(* IEC 61131-3 sources: Antarbhukti-LLM/DatasetCreation/UpgradesGeneration/test_batch, 10 files *)

(* ---- ACTUATOR_2P_sfc_iter_01_L2_iter_01_upgraded.st ---- *)
PROGRAM SFC_Program
(* Auto-generated by SFCJSONConverter *)

VAR
  InitCycle_active : BOOL := FALSE;
  SafetyCheckInput_active : BOOL := FALSE;
  SafetyError_active : BOOL := FALSE;
  Branch_0_active : BOOL := FALSE;
  Branch_1_active : BOOL := FALSE;
  Branch_2_active : BOOL := FALSE;
  Step_255_active : BOOL := FALSE;
  ApplyOutput_active : BOOL := FALSE;
  TimeoutSafeStop_active : BOOL := FALSE;
  SafetyLog_active : BOOL := FALSE;
  IN : INT := 0;
  TEST : INT := 0;
  ARE : INT := 0;
  CYCLE_TIME : TIME := T#0s;
  SENS : INT := 0;
  SELF_ACT_TIME : TIME := T#0s;
  SELF_ACT_PULSE : TIME := T#0s;
  SELF_ACT_CYCLES : INT := 0;
  OUT : BOOL := FALSE;
  ARO : BOOL := FALSE;
  ARX : INT := 0;
  timer : TIMER;
  pwgen : PWGEN;
  INPUT_VALID : BOOL := FALSE;
  SAFETY_ERROR_FLAG : BOOL := FALSE;
  SAFETY_ERROR_CODE : UINT := 0;
  CUMULATIVE_CYCLE_TIME : TIME := T#0s;
  MAX_SAFE_CYCLE_TIME : TIME := T#0s;
  TIMEOUT_EXCEEDED : BOOL := FALSE;
  TIMEOUT_ERROR_FLAG : BOOL := FALSE;
  TIMEOUT_LOG_TIME : TIME := T#0s;
  SAFETY_LOG_CODE : UINT := 0;
  TIMEOUT_LOG_CODE : UINT := 0;
  LOGGED_CYCLE_TIME : TIME := T#0s;
END_VAR

(* --- Initialize initial step --- *)
IF NOT InitCycle_active THEN
  InitCycle_active := TRUE;
END_IF;

(* --- Step actions --- *)
IF InitCycle_active THEN
  timer(trun := MUL_T_AI(SELF_ACT_PULSE,2 * SELF_ACT_CYCLES), toff := SELF_ACT_TIME, Test := TEST, ARE := ARE, arx := ARX); ARX := timer.ARX; ARO := timer.ARO;
END_IF;
IF SafetyCheckInput_active THEN
  INPUT_VALID := (IN >= BYTE#0) AND (IN <= BYTE#255) AND (SENS > BYTE#0) AND (SENS <= BYTE#255); CUMULATIVE_CYCLE_TIME := CUMULATIVE_CYCLE_TIME + CYCLE_TIME;
END_IF;
IF SafetyError_active THEN
  out := FALSE; SAFETY_ERROR_FLAG := TRUE; SAFETY_ERROR_CODE := UINT#1001;
END_IF;
IF Branch_0_active THEN
  pwgen(PTL := SELF_ACT_PULSE, PTH := SELF_ACT_PULSE); out := pwgen.Q;
END_IF;
IF Branch_1_active THEN
  out := FALSE;
END_IF;
IF Branch_2_active THEN
  out := TRUE;
END_IF;
IF Step_255_active THEN
  pwgen.PTH := (CYCLE_TIME * BYTE_TO_TIME(BAND_B(IN,SENS)) ) / BYTE_TO_TIME(BYTE#255); pwgen.PTL := CYCLE_TIME - pwgen.PTH; pwgen(); out := pwgen.Q;
END_IF;
IF ApplyOutput_active THEN
  TIMEOUT_EXCEEDED := CUMULATIVE_CYCLE_TIME > MAX_SAFE_CYCLE_TIME;
END_IF;
IF TimeoutSafeStop_active THEN
  out := FALSE; TIMEOUT_ERROR_FLAG := TRUE; TIMEOUT_LOG_TIME := CUMULATIVE_CYCLE_TIME; CUMULATIVE_CYCLE_TIME := T#0s;
END_IF;
IF SafetyLog_active THEN
  SAFETY_LOG_CODE := SAFETY_ERROR_CODE; TIMEOUT_LOG_CODE := TIMEOUT_ERROR_FLAG; LOGGED_CYCLE_TIME := CUMULATIVE_CYCLE_TIME;
END_IF;

(* --- Transitions --- *)
IF InitCycle_active AND (TRUE) THEN
  InitCycle_active := FALSE;
  SafetyCheckInput_active := TRUE;
END_IF;
IF SafetyCheckInput_active AND (INPUT_VALID = FALSE) THEN
  SafetyCheckInput_active := FALSE;
  SafetyError_active := TRUE;
END_IF;
IF SafetyCheckInput_active AND (INPUT_VALID = TRUE AND aro = TRUE) THEN
  SafetyCheckInput_active := FALSE;
  Branch_0_active := TRUE;
END_IF;
IF SafetyCheckInput_active AND (INPUT_VALID = TRUE AND aro = FALSE AND in<sens) THEN
  SafetyCheckInput_active := FALSE;
  Branch_1_active := TRUE;
END_IF;
IF SafetyCheckInput_active AND (INPUT_VALID = TRUE AND aro = FALSE AND NOT (in<sens) AND BYTE_TO_USINT(in)>USINT#255-BYTE_TO_USINT(sens)) THEN
  SafetyCheckInput_active := FALSE;
  Branch_2_active := TRUE;
END_IF;
IF SafetyCheckInput_active AND (INPUT_VALID = TRUE AND aro = FALSE AND NOT (in<sens) AND NOT (BYTE_TO_USINT(in)>USINT#255-BYTE_TO_USINT(sens))) THEN
  SafetyCheckInput_active := FALSE;
  Step_255_active := TRUE;
END_IF;
IF Branch_0_active AND (TRUE) THEN
  Branch_0_active := FALSE;
  ApplyOutput_active := TRUE;
END_IF;
IF Branch_1_active AND (TRUE) THEN
  Branch_1_active := FALSE;
  ApplyOutput_active := TRUE;
END_IF;
IF Branch_2_active AND (TRUE) THEN
  Branch_2_active := FALSE;
  ApplyOutput_active := TRUE;
END_IF;
IF Step_255_active AND (TRUE) THEN
  Step_255_active := FALSE;
  ApplyOutput_active := TRUE;
END_IF;
IF ApplyOutput_active AND (TIMEOUT_EXCEEDED = TRUE) THEN
  ApplyOutput_active := FALSE;
  TimeoutSafeStop_active := TRUE;
END_IF;
IF ApplyOutput_active AND (TIMEOUT_EXCEEDED = FALSE) THEN
  ApplyOutput_active := FALSE;
  InitCycle_active := TRUE;
END_IF;
IF TimeoutSafeStop_active AND (TRUE) THEN
  TimeoutSafeStop_active := FALSE;
  SafetyLog_active := TRUE;
END_IF;
IF SafetyError_active AND (TRUE) THEN
  SafetyError_active := FALSE;
  SafetyLog_active := TRUE;
END_IF;
IF SafetyLog_active AND (TRUE) THEN
  SafetyLog_active := FALSE;
  InitCycle_active := TRUE;
END_IF;

END_PROGRAM

(* ---- ACTUATOR_2P_sfc_iter_01_L2_iter_02_upgraded.st ---- *)
PROGRAM SFC_Program
(* Auto-generated by SFCJSONConverter *)

VAR
  InitCycle_active : BOOL := FALSE;
  SafetyCheckInput_active : BOOL := FALSE;
  SafetyError_active : BOOL := FALSE;
  SafetyLog_Error_active : BOOL := FALSE;
  Branch_0_active : BOOL := FALSE;
  Branch_1_active : BOOL := FALSE;
  Branch_2_active : BOOL := FALSE;
  Step_255_active : BOOL := FALSE;
  ApplyOutput_active : BOOL := FALSE;
  TimeoutSafeStop_active : BOOL := FALSE;
  SafetyLog_Timeout_active : BOOL := FALSE;
  IN : INT := 0;
  TEST : INT := 0;
  ARE : INT := 0;
  CYCLE_TIME : TIME := T#0s;
  SENS : INT := 0;
  SELF_ACT_TIME : TIME := T#0s;
  SELF_ACT_PULSE : TIME := T#0s;
  SELF_ACT_CYCLES : INT := 0;
  OUT : BOOL := FALSE;
  ARO : BOOL := FALSE;
  ARX : INT := 0;
  timer : TIMER;
  pwgen : PWGEN;
  INPUT_VALID : BOOL := FALSE;
  SAFETY_ERROR_FLAG : BOOL := FALSE;
  SAFETY_ERROR_CODE : UINT := 0;
  CUMULATIVE_CYCLE_TIME : TIME := T#0s;
  MAX_SAFE_CYCLE_TIME : TIME := T#0s;
  TIMEOUT_EXCEEDED : BOOL := FALSE;
  TIMEOUT_ERROR_FLAG : BOOL := FALSE;
  TIMEOUT_LOG_TIME : TIME := T#0s;
  SAFETY_LOG_CODE : UINT := 0;
  SAFETY_LOG_TIME : TIME := T#0s;
  SAFETY_LOG_IN : INT := 0;
  SAFETY_LOG_SENS : INT := 0;
END_VAR

(* --- Initialize initial step --- *)
IF NOT InitCycle_active THEN
  InitCycle_active := TRUE;
END_IF;

(* --- Step actions --- *)
IF InitCycle_active THEN
  timer(trun := MUL_T_AI(SELF_ACT_PULSE,2 * SELF_ACT_CYCLES), toff := SELF_ACT_TIME, Test := TEST, ARE := ARE, arx := ARX); ARX := timer.ARX; ARO := timer.ARO;
END_IF;
IF SafetyCheckInput_active THEN
  INPUT_VALID := (IN >= BYTE#0) AND (IN <= BYTE#255) AND (SENS > BYTE#0) AND (SENS <= BYTE#255); CUMULATIVE_CYCLE_TIME := CUMULATIVE_CYCLE_TIME + CYCLE_TIME;
END_IF;
IF SafetyError_active THEN
  out := FALSE; SAFETY_ERROR_FLAG := TRUE; SAFETY_ERROR_CODE := UINT#1001;
END_IF;
IF SafetyLog_Error_active THEN
  SAFETY_LOG_CODE := SAFETY_ERROR_CODE; SAFETY_LOG_TIME := CUMULATIVE_CYCLE_TIME; SAFETY_LOG_IN := IN; SAFETY_LOG_SENS := SENS;
END_IF;
IF Branch_0_active THEN
  pwgen(PTL := SELF_ACT_PULSE, PTH := SELF_ACT_PULSE); out := pwgen.Q;
END_IF;
IF Branch_1_active THEN
  out := FALSE;
END_IF;
IF Branch_2_active THEN
  out := TRUE;
END_IF;
IF Step_255_active THEN
  pwgen.PTH := (CYCLE_TIME * BYTE_TO_TIME(BAND_B(IN,SENS)) ) / BYTE_TO_TIME(BYTE#255); pwgen.PTL := CYCLE_TIME - pwgen.PTH; pwgen(); out := pwgen.Q;
END_IF;
IF ApplyOutput_active THEN
  TIMEOUT_EXCEEDED := CUMULATIVE_CYCLE_TIME > MAX_SAFE_CYCLE_TIME;
END_IF;
IF TimeoutSafeStop_active THEN
  out := FALSE; TIMEOUT_ERROR_FLAG := TRUE; TIMEOUT_LOG_TIME := CUMULATIVE_CYCLE_TIME; CUMULATIVE_CYCLE_TIME := T#0s;
END_IF;
IF SafetyLog_Timeout_active THEN
  SAFETY_LOG_CODE := UINT#2001; SAFETY_LOG_TIME := TIMEOUT_LOG_TIME;
END_IF;

(* --- Transitions --- *)
IF InitCycle_active AND (TRUE) THEN
  InitCycle_active := FALSE;
  SafetyCheckInput_active := TRUE;
END_IF;
IF SafetyCheckInput_active AND (INPUT_VALID = FALSE) THEN
  SafetyCheckInput_active := FALSE;
  SafetyError_active := TRUE;
END_IF;
IF SafetyCheckInput_active AND (INPUT_VALID = TRUE AND aro = TRUE) THEN
  SafetyCheckInput_active := FALSE;
  Branch_0_active := TRUE;
END_IF;
IF SafetyCheckInput_active AND (INPUT_VALID = TRUE AND aro = FALSE AND in<sens) THEN
  SafetyCheckInput_active := FALSE;
  Branch_1_active := TRUE;
END_IF;
IF SafetyCheckInput_active AND (INPUT_VALID = TRUE AND aro = FALSE AND NOT (in<sens) AND BYTE_TO_USINT(in)>USINT#255-BYTE_TO_USINT(sens)) THEN
  SafetyCheckInput_active := FALSE;
  Branch_2_active := TRUE;
END_IF;
IF SafetyCheckInput_active AND (INPUT_VALID = TRUE AND aro = FALSE AND NOT (in<sens) AND NOT (BYTE_TO_USINT(in)>USINT#255-BYTE_TO_USINT(sens))) THEN
  SafetyCheckInput_active := FALSE;
  Step_255_active := TRUE;
END_IF;
IF Branch_0_active AND (TRUE) THEN
  Branch_0_active := FALSE;
  ApplyOutput_active := TRUE;
END_IF;
IF Branch_1_active AND (TRUE) THEN
  Branch_1_active := FALSE;
  ApplyOutput_active := TRUE;
END_IF;
IF Branch_2_active AND (TRUE) THEN
  Branch_2_active := FALSE;
  ApplyOutput_active := TRUE;
END_IF;
IF Step_255_active AND (TRUE) THEN
  Step_255_active := FALSE;
  ApplyOutput_active := TRUE;
END_IF;
IF ApplyOutput_active AND (TIMEOUT_EXCEEDED = TRUE) THEN
  ApplyOutput_active := FALSE;
  TimeoutSafeStop_active := TRUE;
END_IF;
IF ApplyOutput_active AND (TIMEOUT_EXCEEDED = FALSE) THEN
  ApplyOutput_active := FALSE;
  InitCycle_active := TRUE;
END_IF;
IF TimeoutSafeStop_active AND (TRUE) THEN
  TimeoutSafeStop_active := FALSE;
  SafetyLog_Timeout_active := TRUE;
END_IF;
IF SafetyLog_Timeout_active AND (TRUE) THEN
  SafetyLog_Timeout_active := FALSE;
  InitCycle_active := TRUE;
END_IF;
IF SafetyError_active AND (TRUE) THEN
  SafetyError_active := FALSE;
  SafetyLog_Error_active := TRUE;
END_IF;
IF SafetyLog_Error_active AND (TRUE) THEN
  SafetyLog_Error_active := FALSE;
  SafetyLog_Error_active := TRUE;
END_IF;

END_PROGRAM

(* ---- ACTUATOR_2P_sfc_iter_01_L2_iter_03_upgraded.st ---- *)
PROGRAM SFC_Program
(* Auto-generated by SFCJSONConverter *)

VAR
  InitCycle_active : BOOL := FALSE;
  SafetyCheckInput_active : BOOL := FALSE;
  SafetyLog_active : BOOL := FALSE;
  SafetyError_active : BOOL := FALSE;
  SafetyErrorLog_active : BOOL := FALSE;
  Branch_0_active : BOOL := FALSE;
  Branch_1_active : BOOL := FALSE;
  Branch_2_active : BOOL := FALSE;
  Step_255_active : BOOL := FALSE;
  ApplyOutput_active : BOOL := FALSE;
  TimeoutSafeStop_active : BOOL := FALSE;
  IN : INT := 0;
  TEST : INT := 0;
  ARE : INT := 0;
  CYCLE_TIME : TIME := T#0s;
  SENS : INT := 0;
  SELF_ACT_TIME : TIME := T#0s;
  SELF_ACT_PULSE : TIME := T#0s;
  SELF_ACT_CYCLES : INT := 0;
  OUT : BOOL := FALSE;
  ARO : BOOL := FALSE;
  ARX : INT := 0;
  timer : TIMER;
  pwgen : PWGEN;
  INPUT_VALID : BOOL := FALSE;
  SAFETY_ERROR_FLAG : BOOL := FALSE;
  SAFETY_ERROR_CODE : UINT := 0;
  CUMULATIVE_CYCLE_TIME : TIME := T#0s;
  MAX_SAFE_CYCLE_TIME : TIME := T#0s;
  TIMEOUT_EXCEEDED : BOOL := FALSE;
  TIMEOUT_ERROR_FLAG : BOOL := FALSE;
  TIMEOUT_LOG_TIME : TIME := T#0s;
  SAFETY_LOG_IN : INT := 0;
  SAFETY_LOG_SENS : INT := 0;
  SAFETY_LOG_CUMULATIVE_TIME : TIME := T#0s;
  SAFETY_ERROR_LOG_CODE : UINT := 0;
  SAFETY_ERROR_LOG_TIME : TIME := T#0s;
END_VAR

(* --- Initialize initial step --- *)
IF NOT InitCycle_active THEN
  InitCycle_active := TRUE;
END_IF;

(* --- Step actions --- *)
IF InitCycle_active THEN
  timer(trun := MUL_T_AI(SELF_ACT_PULSE,2 * SELF_ACT_CYCLES), toff := SELF_ACT_TIME, Test := TEST, ARE := ARE, arx := ARX); ARX := timer.ARX; ARO := timer.ARO;
END_IF;
IF SafetyCheckInput_active THEN
  INPUT_VALID := (IN >= BYTE#0) AND (IN <= BYTE#255) AND (SENS > BYTE#0) AND (SENS <= BYTE#255); CUMULATIVE_CYCLE_TIME := CUMULATIVE_CYCLE_TIME + CYCLE_TIME;
END_IF;
IF SafetyLog_active THEN
  SAFETY_LOG_IN := IN; SAFETY_LOG_SENS := SENS; SAFETY_LOG_CUMULATIVE_TIME := CUMULATIVE_CYCLE_TIME;
END_IF;
IF SafetyError_active THEN
  out := FALSE; SAFETY_ERROR_FLAG := TRUE; SAFETY_ERROR_CODE := UINT#1001;
END_IF;
IF SafetyErrorLog_active THEN
  SAFETY_ERROR_LOG_CODE := SAFETY_ERROR_CODE; SAFETY_ERROR_LOG_TIME := CUMULATIVE_CYCLE_TIME;
END_IF;
IF Branch_0_active THEN
  pwgen(PTL := SELF_ACT_PULSE, PTH := SELF_ACT_PULSE); out := pwgen.Q;
END_IF;
IF Branch_1_active THEN
  out := FALSE;
END_IF;
IF Branch_2_active THEN
  out := TRUE;
END_IF;
IF Step_255_active THEN
  pwgen.PTH := (CYCLE_TIME * BYTE_TO_TIME(BAND_B(IN,SENS)) ) / BYTE_TO_TIME(BYTE#255); pwgen.PTL := CYCLE_TIME - pwgen.PTH; pwgen(); out := pwgen.Q;
END_IF;
IF ApplyOutput_active THEN
  TIMEOUT_EXCEEDED := CUMULATIVE_CYCLE_TIME > MAX_SAFE_CYCLE_TIME;
END_IF;
IF TimeoutSafeStop_active THEN
  out := FALSE; TIMEOUT_ERROR_FLAG := TRUE; TIMEOUT_LOG_TIME := CUMULATIVE_CYCLE_TIME; CUMULATIVE_CYCLE_TIME := T#0s;
END_IF;

(* --- Transitions --- *)
IF InitCycle_active AND (TRUE) THEN
  InitCycle_active := FALSE;
  SafetyCheckInput_active := TRUE;
END_IF;
IF SafetyCheckInput_active AND (INPUT_VALID = TRUE) THEN
  SafetyCheckInput_active := FALSE;
  SafetyLog_active := TRUE;
END_IF;
IF SafetyCheckInput_active AND (INPUT_VALID = FALSE) THEN
  SafetyCheckInput_active := FALSE;
  SafetyError_active := TRUE;
END_IF;
IF SafetyLog_active AND (aro = TRUE) THEN
  SafetyLog_active := FALSE;
  Branch_0_active := TRUE;
END_IF;
IF SafetyLog_active AND (aro = FALSE AND in<sens) THEN
  SafetyLog_active := FALSE;
  Branch_1_active := TRUE;
END_IF;
IF SafetyLog_active AND (aro = FALSE AND NOT (in<sens) AND BYTE_TO_USINT(in)>USINT#255-BYTE_TO_USINT(sens)) THEN
  SafetyLog_active := FALSE;
  Branch_2_active := TRUE;
END_IF;
IF SafetyLog_active AND (aro = FALSE AND NOT (in<sens) AND NOT (BYTE_TO_USINT(in)>USINT#255-BYTE_TO_USINT(sens))) THEN
  SafetyLog_active := FALSE;
  Step_255_active := TRUE;
END_IF;
IF Branch_0_active AND (TRUE) THEN
  Branch_0_active := FALSE;
  ApplyOutput_active := TRUE;
END_IF;
IF Branch_1_active AND (TRUE) THEN
  Branch_1_active := FALSE;
  ApplyOutput_active := TRUE;
END_IF;
IF Branch_2_active AND (TRUE) THEN
  Branch_2_active := FALSE;
  ApplyOutput_active := TRUE;
END_IF;
IF Step_255_active AND (TRUE) THEN
  Step_255_active := FALSE;
  ApplyOutput_active := TRUE;
END_IF;
IF ApplyOutput_active AND (TIMEOUT_EXCEEDED = TRUE) THEN
  ApplyOutput_active := FALSE;
  TimeoutSafeStop_active := TRUE;
END_IF;
IF ApplyOutput_active AND (TIMEOUT_EXCEEDED = FALSE) THEN
  ApplyOutput_active := FALSE;
  InitCycle_active := TRUE;
END_IF;
IF TimeoutSafeStop_active AND (TRUE) THEN
  TimeoutSafeStop_active := FALSE;
  InitCycle_active := TRUE;
END_IF;
IF SafetyError_active AND (TRUE) THEN
  SafetyError_active := FALSE;
  SafetyErrorLog_active := TRUE;
END_IF;
IF SafetyErrorLog_active AND (TRUE) THEN
  SafetyErrorLog_active := FALSE;
  SafetyError_active := TRUE;
END_IF;

END_PROGRAM

(* ---- ACTUATOR_2P_sfc_iter_01_upgraded.st ---- *)
PROGRAM SFC_Program
(* Auto-generated by SFCJSONConverter *)

VAR
  InitCycle_active : BOOL := FALSE;
  SafetyCheckInput_active : BOOL := FALSE;
  SafetyError_active : BOOL := FALSE;
  Branch_0_active : BOOL := FALSE;
  Branch_1_active : BOOL := FALSE;
  Branch_2_active : BOOL := FALSE;
  Step_255_active : BOOL := FALSE;
  ApplyOutput_active : BOOL := FALSE;
  TimeoutSafeStop_active : BOOL := FALSE;
  IN : INT := 0;
  TEST : INT := 0;
  ARE : INT := 0;
  CYCLE_TIME : TIME := T#0s;
  SENS : INT := 0;
  SELF_ACT_TIME : TIME := T#0s;
  SELF_ACT_PULSE : TIME := T#0s;
  SELF_ACT_CYCLES : INT := 0;
  OUT : BOOL := FALSE;
  ARO : BOOL := FALSE;
  ARX : INT := 0;
  timer : TIMER;
  pwgen : PWGEN;
  INPUT_VALID : BOOL := FALSE;
  SAFETY_ERROR_FLAG : BOOL := FALSE;
  SAFETY_ERROR_CODE : UINT := 0;
  CUMULATIVE_CYCLE_TIME : TIME := T#0s;
  MAX_SAFE_CYCLE_TIME : TIME := T#0s;
  TIMEOUT_EXCEEDED : BOOL := FALSE;
  TIMEOUT_ERROR_FLAG : BOOL := FALSE;
  TIMEOUT_LOG_TIME : TIME := T#0s;
END_VAR

(* --- Initialize initial step --- *)
IF NOT InitCycle_active THEN
  InitCycle_active := TRUE;
END_IF;

(* --- Step actions --- *)
IF InitCycle_active THEN
  timer(trun := MUL_T_AI(SELF_ACT_PULSE,2 * SELF_ACT_CYCLES), toff := SELF_ACT_TIME, Test := TEST, ARE := ARE, arx := ARX); ARX := timer.ARX; ARO := timer.ARO;
END_IF;
IF SafetyCheckInput_active THEN
  INPUT_VALID := (IN >= BYTE#0) AND (IN <= BYTE#255) AND (SENS > BYTE#0) AND (SENS <= BYTE#255); CUMULATIVE_CYCLE_TIME := CUMULATIVE_CYCLE_TIME + CYCLE_TIME;
END_IF;
IF SafetyError_active THEN
  out := FALSE; SAFETY_ERROR_FLAG := TRUE; SAFETY_ERROR_CODE := UINT#1001;
END_IF;
IF Branch_0_active THEN
  pwgen(PTL := SELF_ACT_PULSE, PTH := SELF_ACT_PULSE); out := pwgen.Q;
END_IF;
IF Branch_1_active THEN
  out := FALSE;
END_IF;
IF Branch_2_active THEN
  out := TRUE;
END_IF;
IF Step_255_active THEN
  pwgen.PTH := (CYCLE_TIME * BYTE_TO_TIME(BAND_B(IN,SENS)) ) / BYTE_TO_TIME(BYTE#255); pwgen.PTL := CYCLE_TIME - pwgen.PTH; pwgen(); out := pwgen.Q;
END_IF;
IF ApplyOutput_active THEN
  TIMEOUT_EXCEEDED := CUMULATIVE_CYCLE_TIME > MAX_SAFE_CYCLE_TIME;
END_IF;
IF TimeoutSafeStop_active THEN
  out := FALSE; TIMEOUT_ERROR_FLAG := TRUE; TIMEOUT_LOG_TIME := CUMULATIVE_CYCLE_TIME; CUMULATIVE_CYCLE_TIME := T#0s;
END_IF;

(* --- Transitions --- *)
IF InitCycle_active AND (TRUE) THEN
  InitCycle_active := FALSE;
  SafetyCheckInput_active := TRUE;
END_IF;
IF SafetyCheckInput_active AND (INPUT_VALID = FALSE) THEN
  SafetyCheckInput_active := FALSE;
  SafetyError_active := TRUE;
END_IF;
IF SafetyCheckInput_active AND (INPUT_VALID = TRUE AND aro = TRUE) THEN
  SafetyCheckInput_active := FALSE;
  Branch_0_active := TRUE;
END_IF;
IF SafetyCheckInput_active AND (INPUT_VALID = TRUE AND aro = FALSE AND in<sens) THEN
  SafetyCheckInput_active := FALSE;
  Branch_1_active := TRUE;
END_IF;
IF SafetyCheckInput_active AND (INPUT_VALID = TRUE AND aro = FALSE AND NOT (in<sens) AND BYTE_TO_USINT(in)>USINT#255-BYTE_TO_USINT(sens)) THEN
  SafetyCheckInput_active := FALSE;
  Branch_2_active := TRUE;
END_IF;
IF SafetyCheckInput_active AND (INPUT_VALID = TRUE AND aro = FALSE AND NOT (in<sens) AND NOT (BYTE_TO_USINT(in)>USINT#255-BYTE_TO_USINT(sens))) THEN
  SafetyCheckInput_active := FALSE;
  Step_255_active := TRUE;
END_IF;
IF Branch_0_active AND (TRUE) THEN
  Branch_0_active := FALSE;
  ApplyOutput_active := TRUE;
END_IF;
IF Branch_1_active AND (TRUE) THEN
  Branch_1_active := FALSE;
  ApplyOutput_active := TRUE;
END_IF;
IF Branch_2_active AND (TRUE) THEN
  Branch_2_active := FALSE;
  ApplyOutput_active := TRUE;
END_IF;
IF Step_255_active AND (TRUE) THEN
  Step_255_active := FALSE;
  ApplyOutput_active := TRUE;
END_IF;
IF ApplyOutput_active AND (TIMEOUT_EXCEEDED = TRUE) THEN
  ApplyOutput_active := FALSE;
  TimeoutSafeStop_active := TRUE;
END_IF;
IF ApplyOutput_active AND (TIMEOUT_EXCEEDED = FALSE) THEN
  ApplyOutput_active := FALSE;
  InitCycle_active := TRUE;
END_IF;
IF TimeoutSafeStop_active AND (TRUE) THEN
  TimeoutSafeStop_active := FALSE;
  InitCycle_active := TRUE;
END_IF;
IF SafetyError_active AND (TRUE) THEN
  SafetyError_active := FALSE;
  SafetyError_active := TRUE;
END_IF;

END_PROGRAM

(* ---- ACTUATOR_2P_sfc_iter_02_L2_iter_01_upgraded.st ---- *)
PROGRAM SFC_Program
(* Auto-generated by SFCJSONConverter *)

VAR
  InitCycle_active : BOOL := FALSE;
  SafetyCheckInput_active : BOOL := FALSE;
  SafetyError_active : BOOL := FALSE;
  TimeoutSafeStop_active : BOOL := FALSE;
  Branch_0_active : BOOL := FALSE;
  Branch_1_active : BOOL := FALSE;
  Branch_2_active : BOOL := FALSE;
  SensZeroCheck_active : BOOL := FALSE;
  SensZeroSafeState_active : BOOL := FALSE;
  Step_255_active : BOOL := FALSE;
  ApplyOutput_active : BOOL := FALSE;
  SafetyLog_active : BOOL := FALSE;
  IN : INT := 0;
  TEST : INT := 0;
  ARE : INT := 0;
  CYCLE_TIME : TIME := T#0s;
  SENS : INT := 0;
  SELF_ACT_TIME : TIME := T#0s;
  SELF_ACT_PULSE : TIME := T#0s;
  SELF_ACT_CYCLES : INT := 0;
  OUT : BOOL := FALSE;
  ARO : BOOL := FALSE;
  ARX : INT := 0;
  timer : TIMER;
  pwgen : PWGEN;
  INPUT_VALID : BOOL := FALSE;
  TIMEOUT_EXCEEDED : BOOL := FALSE;
  CYCLE_ELAPSED_TIME : TIME := T#0s;
  MAX_SAFE_CYCLE_TIME : TIME := T#0s;
  SCAN_TIME : TIME := T#0s;
  SAFETY_ERROR_FLAG : BOOL := FALSE;
  TIMEOUT_ERROR_FLAG : BOOL := FALSE;
  SENS_ZERO_ERROR : BOOL := FALSE;
  SENS_ZERO_FLAG : BOOL := FALSE;
  SAFETY_LOG_TIME : TIME := T#0s;
  SAFETY_LOG_ERROR : BOOL := FALSE;
END_VAR

(* --- Initialize initial step --- *)
IF NOT InitCycle_active THEN
  InitCycle_active := TRUE;
END_IF;

(* --- Step actions --- *)
IF InitCycle_active THEN
  timer(trun := MUL_T_AI(SELF_ACT_PULSE,2 * SELF_ACT_CYCLES), toff := SELF_ACT_TIME, Test := TEST, ARE := ARE, arx := ARX); ARX := timer.ARX; ARO := timer.ARO; CYCLE_ELAPSED_TIME := CYCLE_ELAPSED_TIME + SCAN_TIME;
END_IF;
IF SafetyCheckInput_active THEN
  INPUT_VALID := (IN >= BYTE#0) AND (IN <= BYTE#255) AND (SENS > BYTE#0) AND (SENS <= BYTE#255); TIMEOUT_EXCEEDED := CYCLE_ELAPSED_TIME > MAX_SAFE_CYCLE_TIME;
END_IF;
IF SafetyError_active THEN
  OUT := FALSE; SAFETY_ERROR_FLAG := TRUE; ARO := FALSE;
END_IF;
IF TimeoutSafeStop_active THEN
  OUT := FALSE; TIMEOUT_ERROR_FLAG := TRUE; ARO := FALSE;
END_IF;
IF Branch_0_active THEN
  pwgen(PTL := SELF_ACT_PULSE, PTH := SELF_ACT_PULSE); out := pwgen.Q;
END_IF;
IF Branch_1_active THEN
  out := FALSE;
END_IF;
IF Branch_2_active THEN
  out := TRUE;
END_IF;
IF SensZeroCheck_active THEN
  SENS_ZERO_ERROR := (SENS == BYTE#0);
END_IF;
IF SensZeroSafeState_active THEN
  OUT := FALSE; SENS_ZERO_FLAG := TRUE;
END_IF;
IF Step_255_active THEN
  pwgen.PTH := (CYCLE_TIME * BYTE_TO_TIME(BAND_B(IN,SENS)) ) / BYTE_TO_TIME(BYTE#255); pwgen.PTL := CYCLE_TIME - pwgen.PTH; pwgen(); out := pwgen.Q;
END_IF;
IF ApplyOutput_active THEN
  CYCLE_ELAPSED_TIME := TIME#0s;
END_IF;
IF SafetyLog_active THEN
  SAFETY_LOG_TIME := CYCLE_ELAPSED_TIME; SAFETY_LOG_ERROR := SAFETY_ERROR_FLAG OR TIMEOUT_ERROR_FLAG OR SENS_ZERO_FLAG;
END_IF;

(* --- Transitions --- *)
IF InitCycle_active AND (TRUE) THEN
  InitCycle_active := FALSE;
  SafetyCheckInput_active := TRUE;
END_IF;
IF SafetyCheckInput_active AND (INPUT_VALID = FALSE) THEN
  SafetyCheckInput_active := FALSE;
  SafetyError_active := TRUE;
END_IF;
IF SafetyCheckInput_active AND (INPUT_VALID = TRUE AND TIMEOUT_EXCEEDED = TRUE) THEN
  SafetyCheckInput_active := FALSE;
  TimeoutSafeStop_active := TRUE;
END_IF;
IF SafetyCheckInput_active AND (INPUT_VALID = TRUE AND TIMEOUT_EXCEEDED = FALSE AND aro = TRUE) THEN
  SafetyCheckInput_active := FALSE;
  Branch_0_active := TRUE;
END_IF;
IF SafetyCheckInput_active AND (INPUT_VALID = TRUE AND TIMEOUT_EXCEEDED = FALSE AND aro = FALSE AND in<sens) THEN
  SafetyCheckInput_active := FALSE;
  Branch_1_active := TRUE;
END_IF;
IF SafetyCheckInput_active AND (INPUT_VALID = TRUE AND TIMEOUT_EXCEEDED = FALSE AND aro = FALSE AND NOT (in<sens) AND BYTE_TO_USINT(in)>USINT#255-BYTE_TO_USINT(sens)) THEN
  SafetyCheckInput_active := FALSE;
  Branch_2_active := TRUE;
END_IF;
IF SafetyCheckInput_active AND (INPUT_VALID = TRUE AND TIMEOUT_EXCEEDED = FALSE AND aro = FALSE AND NOT (in<sens) AND NOT (BYTE_TO_USINT(in)>USINT#255-BYTE_TO_USINT(sens))) THEN
  SafetyCheckInput_active := FALSE;
  SensZeroCheck_active := TRUE;
END_IF;
IF SensZeroCheck_active AND (SENS_ZERO_ERROR = TRUE) THEN
  SensZeroCheck_active := FALSE;
  SensZeroSafeState_active := TRUE;
END_IF;
IF SensZeroCheck_active AND (SENS_ZERO_ERROR = FALSE) THEN
  SensZeroCheck_active := FALSE;
  Step_255_active := TRUE;
END_IF;
IF Branch_0_active AND (TRUE) THEN
  Branch_0_active := FALSE;
  ApplyOutput_active := TRUE;
END_IF;
IF Branch_1_active AND (TRUE) THEN
  Branch_1_active := FALSE;
  ApplyOutput_active := TRUE;
END_IF;
IF Branch_2_active AND (TRUE) THEN
  Branch_2_active := FALSE;
  ApplyOutput_active := TRUE;
END_IF;
IF Step_255_active AND (TRUE) THEN
  Step_255_active := FALSE;
  ApplyOutput_active := TRUE;
END_IF;
IF SensZeroSafeState_active AND (TRUE) THEN
  SensZeroSafeState_active := FALSE;
  SafetyLog_active := TRUE;
END_IF;
IF SafetyError_active AND (TRUE) THEN
  SafetyError_active := FALSE;
  SafetyLog_active := TRUE;
END_IF;
IF TimeoutSafeStop_active AND (TRUE) THEN
  TimeoutSafeStop_active := FALSE;
  SafetyLog_active := TRUE;
END_IF;
IF SafetyLog_active AND (TRUE) THEN
  SafetyLog_active := FALSE;
  InitCycle_active := TRUE;
END_IF;
IF ApplyOutput_active AND (TRUE) THEN
  ApplyOutput_active := FALSE;
  InitCycle_active := TRUE;
END_IF;

END_PROGRAM

(* ---- ACTUATOR_2P_sfc_iter_02_L2_iter_02_upgraded.st ---- *)
PROGRAM SFC_Program
(* Auto-generated by SFCJSONConverter *)

VAR
  InitCycle_active : BOOL := FALSE;
  SafetyCheckInput_active : BOOL := FALSE;
  SafetyError_active : BOOL := FALSE;
  TimeoutSafeStop_active : BOOL := FALSE;
  Branch_0_active : BOOL := FALSE;
  Branch_1_active : BOOL := FALSE;
  Branch_2_active : BOOL := FALSE;
  Step_255_active : BOOL := FALSE;
  ApplyOutput_active : BOOL := FALSE;
  DivZeroSafeStop_active : BOOL := FALSE;
  InvalidCycleTimeStop_active : BOOL := FALSE;
  IN : INT := 0;
  TEST : INT := 0;
  ARE : INT := 0;
  CYCLE_TIME : TIME := T#0s;
  SENS : INT := 0;
  SELF_ACT_TIME : TIME := T#0s;
  SELF_ACT_PULSE : TIME := T#0s;
  SELF_ACT_CYCLES : INT := 0;
  OUT : BOOL := FALSE;
  ARO : BOOL := FALSE;
  ARX : INT := 0;
  timer : TIMER;
  pwgen : PWGEN;
  INPUT_VALID : BOOL := FALSE;
  TIMEOUT_EXCEEDED : BOOL := FALSE;
  CYCLE_ELAPSED_TIME : TIME := T#0s;
  MAX_SAFE_CYCLE_TIME : TIME := T#0s;
  SCAN_TIME : TIME := T#0s;
  SAFETY_ERROR_FLAG : BOOL := FALSE;
  TIMEOUT_ERROR_FLAG : BOOL := FALSE;
  DIV_ZERO_ERROR_FLAG : BOOL := FALSE;
  CYCLE_TIME_ERROR_FLAG : BOOL := FALSE;
END_VAR

(* --- Initialize initial step --- *)
IF NOT InitCycle_active THEN
  InitCycle_active := TRUE;
END_IF;

(* --- Step actions --- *)
IF InitCycle_active THEN
  timer(trun := MUL_T_AI(SELF_ACT_PULSE,2 * SELF_ACT_CYCLES), toff := SELF_ACT_TIME, Test := TEST, ARE := ARE, arx := ARX); ARX := timer.ARX; ARO := timer.ARO; CYCLE_ELAPSED_TIME := CYCLE_ELAPSED_TIME + SCAN_TIME;
END_IF;
IF SafetyCheckInput_active THEN
  INPUT_VALID := (IN >= BYTE#0) AND (IN <= BYTE#255) AND (SENS > BYTE#0) AND (SENS <= BYTE#255); TIMEOUT_EXCEEDED := CYCLE_ELAPSED_TIME > MAX_SAFE_CYCLE_TIME;
END_IF;
IF SafetyError_active THEN
  OUT := FALSE; SAFETY_ERROR_FLAG := TRUE; ARO := FALSE;
END_IF;
IF TimeoutSafeStop_active THEN
  OUT := FALSE; TIMEOUT_ERROR_FLAG := TRUE; ARO := FALSE;
END_IF;
IF Branch_0_active THEN
  pwgen(PTL := SELF_ACT_PULSE, PTH := SELF_ACT_PULSE); out := pwgen.Q;
END_IF;
IF Branch_1_active THEN
  out := FALSE;
END_IF;
IF Branch_2_active THEN
  out := TRUE;
END_IF;
IF Step_255_active THEN
  pwgen.PTH := (CYCLE_TIME * BYTE_TO_TIME(BAND_B(IN,SENS)) ) / BYTE_TO_TIME(BYTE#255); pwgen.PTL := CYCLE_TIME - pwgen.PTH; pwgen(); out := pwgen.Q;
END_IF;
IF ApplyOutput_active THEN
  CYCLE_ELAPSED_TIME := TIME#0s;
END_IF;
IF DivZeroSafeStop_active THEN
  OUT := FALSE; DIV_ZERO_ERROR_FLAG := TRUE; ARO := FALSE;
END_IF;
IF InvalidCycleTimeStop_active THEN
  OUT := FALSE; CYCLE_TIME_ERROR_FLAG := TRUE; ARO := FALSE;
END_IF;

(* --- Transitions --- *)
IF InitCycle_active AND (TRUE) THEN
  InitCycle_active := FALSE;
  SafetyCheckInput_active := TRUE;
END_IF;
IF SafetyCheckInput_active AND (INPUT_VALID = FALSE) THEN
  SafetyCheckInput_active := FALSE;
  SafetyError_active := TRUE;
END_IF;
IF SafetyCheckInput_active AND (INPUT_VALID = TRUE AND TIMEOUT_EXCEEDED = TRUE) THEN
  SafetyCheckInput_active := FALSE;
  TimeoutSafeStop_active := TRUE;
END_IF;
IF SafetyCheckInput_active AND (INPUT_VALID = TRUE AND TIMEOUT_EXCEEDED = FALSE AND aro = TRUE) THEN
  SafetyCheckInput_active := FALSE;
  Branch_0_active := TRUE;
END_IF;
IF SafetyCheckInput_active AND (INPUT_VALID = TRUE AND TIMEOUT_EXCEEDED = FALSE AND aro = FALSE AND in<sens) THEN
  SafetyCheckInput_active := FALSE;
  Branch_1_active := TRUE;
END_IF;
IF SafetyCheckInput_active AND (INPUT_VALID = TRUE AND TIMEOUT_EXCEEDED = FALSE AND aro = FALSE AND NOT (in<sens) AND BYTE_TO_USINT(in)>USINT#255-BYTE_TO_USINT(sens)) THEN
  SafetyCheckInput_active := FALSE;
  Branch_2_active := TRUE;
END_IF;
IF SafetyCheckInput_active AND (INPUT_VALID = TRUE AND TIMEOUT_EXCEEDED = FALSE AND aro = FALSE AND NOT (in<sens) AND NOT (BYTE_TO_USINT(in)>USINT#255-BYTE_TO_USINT(sens))) THEN
  SafetyCheckInput_active := FALSE;
  Step_255_active := TRUE;
END_IF;
IF Branch_0_active AND (TRUE) THEN
  Branch_0_active := FALSE;
  ApplyOutput_active := TRUE;
END_IF;
IF Branch_1_active AND (TRUE) THEN
  Branch_1_active := FALSE;
  ApplyOutput_active := TRUE;
END_IF;
IF Branch_2_active AND (TRUE) THEN
  Branch_2_active := FALSE;
  ApplyOutput_active := TRUE;
END_IF;
IF Step_255_active AND (TRUE) THEN
  Step_255_active := FALSE;
  ApplyOutput_active := TRUE;
END_IF;
IF ApplyOutput_active AND (TRUE) THEN
  ApplyOutput_active := FALSE;
  InitCycle_active := TRUE;
END_IF;
IF SafetyCheckInput_active AND (INPUT_VALID = TRUE AND TIMEOUT_EXCEEDED = FALSE AND aro = FALSE AND NOT (in<sens) AND NOT (BYTE_TO_USINT(in)>USINT#255-BYTE_TO_USINT(sens)) AND SENS = BYTE#0) THEN
  SafetyCheckInput_active := FALSE;
  DivZeroSafeStop_active := TRUE;
END_IF;
IF SafetyCheckInput_active AND (INPUT_VALID = TRUE AND TIMEOUT_EXCEEDED = FALSE AND aro = FALSE AND NOT (in<sens) AND NOT (BYTE_TO_USINT(in)>USINT#255-BYTE_TO_USINT(sens)) AND CYCLE_TIME <= TIME#0s) THEN
  SafetyCheckInput_active := FALSE;
  InvalidCycleTimeStop_active := TRUE;
END_IF;
IF DivZeroSafeStop_active AND (TRUE) THEN
  DivZeroSafeStop_active := FALSE;
  ApplyOutput_active := TRUE;
END_IF;
IF InvalidCycleTimeStop_active AND (TRUE) THEN
  InvalidCycleTimeStop_active := FALSE;
  ApplyOutput_active := TRUE;
END_IF;

END_PROGRAM

(* ---- ACTUATOR_2P_sfc_iter_02_L2_iter_03_upgraded.st ---- *)
PROGRAM SFC_Program
(* Auto-generated by SFCJSONConverter *)

VAR
  InitCycle_active : BOOL := FALSE;
  SafetyCheckInput_active : BOOL := FALSE;
  ValidateSensInput_active : BOOL := FALSE;
  SensSafetyError_active : BOOL := FALSE;
  SafetyError_active : BOOL := FALSE;
  TimeoutSafeStop_active : BOOL := FALSE;
  Branch_0_active : BOOL := FALSE;
  WatchdogCheck_0_active : BOOL := FALSE;
  WatchdogError_active : BOOL := FALSE;
  Branch_1_active : BOOL := FALSE;
  Branch_2_active : BOOL := FALSE;
  Step_255_active : BOOL := FALSE;
  WatchdogCheck_255_active : BOOL := FALSE;
  ApplyOutput_active : BOOL := FALSE;
  IN : INT := 0;
  TEST : INT := 0;
  ARE : INT := 0;
  CYCLE_TIME : TIME := T#0s;
  SENS : INT := 0;
  SELF_ACT_TIME : TIME := T#0s;
  SELF_ACT_PULSE : TIME := T#0s;
  SELF_ACT_CYCLES : INT := 0;
  OUT : BOOL := FALSE;
  ARO : BOOL := FALSE;
  ARX : INT := 0;
  timer : TIMER;
  pwgen : PWGEN;
  INPUT_VALID : BOOL := FALSE;
  TIMEOUT_EXCEEDED : BOOL := FALSE;
  CYCLE_ELAPSED_TIME : TIME := T#0s;
  MAX_SAFE_CYCLE_TIME : TIME := T#0s;
  SCAN_TIME : TIME := T#0s;
  SAFETY_ERROR_FLAG : BOOL := FALSE;
  TIMEOUT_ERROR_FLAG : BOOL := FALSE;
  SENS_VALID : BOOL := FALSE;
  SENS_ERROR_FLAG : BOOL := FALSE;
  PWGEN_VALID_0 : BOOL := FALSE;
  PWGEN_VALID_255 : BOOL := FALSE;
  WATCHDOG_ERROR_FLAG : BOOL := FALSE;
END_VAR

(* --- Initialize initial step --- *)
IF NOT InitCycle_active THEN
  InitCycle_active := TRUE;
END_IF;

(* --- Step actions --- *)
IF InitCycle_active THEN
  timer(trun := MUL_T_AI(SELF_ACT_PULSE,2 * SELF_ACT_CYCLES), toff := SELF_ACT_TIME, Test := TEST, ARE := ARE, arx := ARX); ARX := timer.ARX; ARO := timer.ARO; CYCLE_ELAPSED_TIME := CYCLE_ELAPSED_TIME + SCAN_TIME;
END_IF;
IF SafetyCheckInput_active THEN
  INPUT_VALID := (IN >= BYTE#0) AND (IN <= BYTE#255) AND (SENS > BYTE#0) AND (SENS <= BYTE#255); TIMEOUT_EXCEEDED := CYCLE_ELAPSED_TIME > MAX_SAFE_CYCLE_TIME;
END_IF;
IF ValidateSensInput_active THEN
  SENS_VALID := (SENS > BYTE#0);
END_IF;
IF SensSafetyError_active THEN
  OUT := FALSE; SAFETY_ERROR_FLAG := TRUE; ARO := FALSE; SENS_ERROR_FLAG := TRUE;
END_IF;
IF SafetyError_active THEN
  OUT := FALSE; SAFETY_ERROR_FLAG := TRUE; ARO := FALSE;
END_IF;
IF TimeoutSafeStop_active THEN
  OUT := FALSE; TIMEOUT_ERROR_FLAG := TRUE; ARO := FALSE;
END_IF;
IF Branch_0_active THEN
  pwgen(PTL := SELF_ACT_PULSE, PTH := SELF_ACT_PULSE); out := pwgen.Q;
END_IF;
IF WatchdogCheck_0_active THEN
  PWGEN_VALID_0 := (pwgen.Q = TRUE) OR (pwgen.Q = FALSE);
END_IF;
IF WatchdogError_active THEN
  OUT := FALSE; WATCHDOG_ERROR_FLAG := TRUE; ARO := FALSE;
END_IF;
IF Branch_1_active THEN
  out := FALSE;
END_IF;
IF Branch_2_active THEN
  out := TRUE;
END_IF;
IF Step_255_active THEN
  pwgen.PTH := (CYCLE_TIME * BYTE_TO_TIME(BAND_B(IN,SENS)) ) / BYTE_TO_TIME(BYTE#255); pwgen.PTL := CYCLE_TIME - pwgen.PTH; pwgen(); out := pwgen.Q;
END_IF;
IF WatchdogCheck_255_active THEN
  PWGEN_VALID_255 := (pwgen.Q = TRUE) OR (pwgen.Q = FALSE);
END_IF;
IF ApplyOutput_active THEN
  CYCLE_ELAPSED_TIME := TIME#0s;
END_IF;

(* --- Transitions --- *)
IF InitCycle_active AND (TRUE) THEN
  InitCycle_active := FALSE;
  SafetyCheckInput_active := TRUE;
END_IF;
IF SafetyCheckInput_active AND (INPUT_VALID = TRUE AND TIMEOUT_EXCEEDED = FALSE) THEN
  SafetyCheckInput_active := FALSE;
  ValidateSensInput_active := TRUE;
END_IF;
IF SafetyCheckInput_active AND (INPUT_VALID = FALSE) THEN
  SafetyCheckInput_active := FALSE;
  SafetyError_active := TRUE;
END_IF;
IF SafetyCheckInput_active AND (INPUT_VALID = TRUE AND TIMEOUT_EXCEEDED = TRUE) THEN
  SafetyCheckInput_active := FALSE;
  TimeoutSafeStop_active := TRUE;
END_IF;
IF ValidateSensInput_active AND (SENS_VALID = FALSE) THEN
  ValidateSensInput_active := FALSE;
  SensSafetyError_active := TRUE;
END_IF;
IF ValidateSensInput_active AND (SENS_VALID = TRUE AND aro = TRUE) THEN
  ValidateSensInput_active := FALSE;
  Branch_0_active := TRUE;
END_IF;
IF ValidateSensInput_active AND (SENS_VALID = TRUE AND aro = FALSE AND in<sens) THEN
  ValidateSensInput_active := FALSE;
  Branch_1_active := TRUE;
END_IF;
IF ValidateSensInput_active AND (SENS_VALID = TRUE AND aro = FALSE AND NOT (in<sens) AND BYTE_TO_USINT(in)>USINT#255-BYTE_TO_USINT(sens)) THEN
  ValidateSensInput_active := FALSE;
  Branch_2_active := TRUE;
END_IF;
IF ValidateSensInput_active AND (SENS_VALID = TRUE AND aro = FALSE AND NOT (in<sens) AND NOT (BYTE_TO_USINT(in)>USINT#255-BYTE_TO_USINT(sens))) THEN
  ValidateSensInput_active := FALSE;
  Step_255_active := TRUE;
END_IF;
IF Branch_0_active AND (TRUE) THEN
  Branch_0_active := FALSE;
  WatchdogCheck_0_active := TRUE;
END_IF;
IF WatchdogCheck_0_active AND (PWGEN_VALID_0 = FALSE) THEN
  WatchdogCheck_0_active := FALSE;
  WatchdogError_active := TRUE;
END_IF;
IF WatchdogCheck_0_active AND (PWGEN_VALID_0 = TRUE) THEN
  WatchdogCheck_0_active := FALSE;
  ApplyOutput_active := TRUE;
END_IF;
IF Branch_1_active AND (TRUE) THEN
  Branch_1_active := FALSE;
  ApplyOutput_active := TRUE;
END_IF;
IF Branch_2_active AND (TRUE) THEN
  Branch_2_active := FALSE;
  ApplyOutput_active := TRUE;
END_IF;
IF Step_255_active AND (TRUE) THEN
  Step_255_active := FALSE;
  WatchdogCheck_255_active := TRUE;
END_IF;
IF WatchdogCheck_255_active AND (PWGEN_VALID_255 = FALSE) THEN
  WatchdogCheck_255_active := FALSE;
  WatchdogError_active := TRUE;
END_IF;
IF WatchdogCheck_255_active AND (PWGEN_VALID_255 = TRUE) THEN
  WatchdogCheck_255_active := FALSE;
  ApplyOutput_active := TRUE;
END_IF;
IF ApplyOutput_active AND (TRUE) THEN
  ApplyOutput_active := FALSE;
  InitCycle_active := TRUE;
END_IF;
IF SensSafetyError_active AND (TRUE) THEN
  SensSafetyError_active := FALSE;
  ApplyOutput_active := TRUE;
END_IF;
IF SafetyError_active AND (TRUE) THEN
  SafetyError_active := FALSE;
  ApplyOutput_active := TRUE;
END_IF;
IF TimeoutSafeStop_active AND (TRUE) THEN
  TimeoutSafeStop_active := FALSE;
  ApplyOutput_active := TRUE;
END_IF;
IF WatchdogError_active AND (TRUE) THEN
  WatchdogError_active := FALSE;
  ApplyOutput_active := TRUE;
END_IF;

END_PROGRAM

(* ---- ACTUATOR_2P_sfc_iter_02_upgraded.st ---- *)
PROGRAM SFC_Program
(* Auto-generated by SFCJSONConverter *)

VAR
  InitCycle_active : BOOL := FALSE;
  SafetyCheckInput_active : BOOL := FALSE;
  SafetyError_active : BOOL := FALSE;
  TimeoutSafeStop_active : BOOL := FALSE;
  Branch_0_active : BOOL := FALSE;
  Branch_1_active : BOOL := FALSE;
  Branch_2_active : BOOL := FALSE;
  Step_255_active : BOOL := FALSE;
  ApplyOutput_active : BOOL := FALSE;
  IN : INT := 0;
  TEST : INT := 0;
  ARE : INT := 0;
  CYCLE_TIME : TIME := T#0s;
  SENS : INT := 0;
  SELF_ACT_TIME : TIME := T#0s;
  SELF_ACT_PULSE : TIME := T#0s;
  SELF_ACT_CYCLES : INT := 0;
  OUT : BOOL := FALSE;
  ARO : BOOL := FALSE;
  ARX : INT := 0;
  timer : TIMER;
  pwgen : PWGEN;
  INPUT_VALID : BOOL := FALSE;
  TIMEOUT_EXCEEDED : BOOL := FALSE;
  CYCLE_ELAPSED_TIME : TIME := T#0s;
  MAX_SAFE_CYCLE_TIME : TIME := T#0s;
  SCAN_TIME : TIME := T#0s;
  SAFETY_ERROR_FLAG : BOOL := FALSE;
  TIMEOUT_ERROR_FLAG : BOOL := FALSE;
END_VAR

(* --- Initialize initial step --- *)
IF NOT InitCycle_active THEN
  InitCycle_active := TRUE;
END_IF;

(* --- Step actions --- *)
IF InitCycle_active THEN
  timer(trun := MUL_T_AI(SELF_ACT_PULSE,2 * SELF_ACT_CYCLES), toff := SELF_ACT_TIME, Test := TEST, ARE := ARE, arx := ARX); ARX := timer.ARX; ARO := timer.ARO; CYCLE_ELAPSED_TIME := CYCLE_ELAPSED_TIME + SCAN_TIME;
END_IF;
IF SafetyCheckInput_active THEN
  INPUT_VALID := (IN >= BYTE#0) AND (IN <= BYTE#255) AND (SENS > BYTE#0) AND (SENS <= BYTE#255); TIMEOUT_EXCEEDED := CYCLE_ELAPSED_TIME > MAX_SAFE_CYCLE_TIME;
END_IF;
IF SafetyError_active THEN
  OUT := FALSE; SAFETY_ERROR_FLAG := TRUE; ARO := FALSE;
END_IF;
IF TimeoutSafeStop_active THEN
  OUT := FALSE; TIMEOUT_ERROR_FLAG := TRUE; ARO := FALSE;
END_IF;
IF Branch_0_active THEN
  pwgen(PTL := SELF_ACT_PULSE, PTH := SELF_ACT_PULSE); out := pwgen.Q;
END_IF;
IF Branch_1_active THEN
  out := FALSE;
END_IF;
IF Branch_2_active THEN
  out := TRUE;
END_IF;
IF Step_255_active THEN
  pwgen.PTH := (CYCLE_TIME * BYTE_TO_TIME(BAND_B(IN,SENS)) ) / BYTE_TO_TIME(BYTE#255); pwgen.PTL := CYCLE_TIME - pwgen.PTH; pwgen(); out := pwgen.Q;
END_IF;
IF ApplyOutput_active THEN
  CYCLE_ELAPSED_TIME := TIME#0s;
END_IF;

(* --- Transitions --- *)
IF InitCycle_active AND (TRUE) THEN
  InitCycle_active := FALSE;
  SafetyCheckInput_active := TRUE;
END_IF;
IF SafetyCheckInput_active AND (INPUT_VALID = FALSE) THEN
  SafetyCheckInput_active := FALSE;
  SafetyError_active := TRUE;
END_IF;
IF SafetyCheckInput_active AND (INPUT_VALID = TRUE AND TIMEOUT_EXCEEDED = TRUE) THEN
  SafetyCheckInput_active := FALSE;
  TimeoutSafeStop_active := TRUE;
END_IF;
IF SafetyCheckInput_active AND (INPUT_VALID = TRUE AND TIMEOUT_EXCEEDED = FALSE AND aro = TRUE) THEN
  SafetyCheckInput_active := FALSE;
  Branch_0_active := TRUE;
END_IF;
IF SafetyCheckInput_active AND (INPUT_VALID = TRUE AND TIMEOUT_EXCEEDED = FALSE AND aro = FALSE AND in<sens) THEN
  SafetyCheckInput_active := FALSE;
  Branch_1_active := TRUE;
END_IF;
IF SafetyCheckInput_active AND (INPUT_VALID = TRUE AND TIMEOUT_EXCEEDED = FALSE AND aro = FALSE AND NOT (in<sens) AND BYTE_TO_USINT(in)>USINT#255-BYTE_TO_USINT(sens)) THEN
  SafetyCheckInput_active := FALSE;
  Branch_2_active := TRUE;
END_IF;
IF SafetyCheckInput_active AND (INPUT_VALID = TRUE AND TIMEOUT_EXCEEDED = FALSE AND aro = FALSE AND NOT (in<sens) AND NOT (BYTE_TO_USINT(in)>USINT#255-BYTE_TO_USINT(sens))) THEN
  SafetyCheckInput_active := FALSE;
  Step_255_active := TRUE;
END_IF;
IF Branch_0_active AND (TRUE) THEN
  Branch_0_active := FALSE;
  ApplyOutput_active := TRUE;
END_IF;
IF Branch_1_active AND (TRUE) THEN
  Branch_1_active := FALSE;
  ApplyOutput_active := TRUE;
END_IF;
IF Branch_2_active AND (TRUE) THEN
  Branch_2_active := FALSE;
  ApplyOutput_active := TRUE;
END_IF;
IF Step_255_active AND (TRUE) THEN
  Step_255_active := FALSE;
  ApplyOutput_active := TRUE;
END_IF;
IF ApplyOutput_active AND (TRUE) THEN
  ApplyOutput_active := FALSE;
  InitCycle_active := TRUE;
END_IF;

END_PROGRAM

(* ---- ACTUATOR_2P_sfc_iter_03_L2_iter_01_upgraded.st ---- *)
PROGRAM SFC_Program
(* Auto-generated by SFCJSONConverter *)

VAR
  InitCycle_active : BOOL := FALSE;
  SafetyCheckInput_active : BOOL := FALSE;
  SafetyError_active : BOOL := FALSE;
  TimeoutSafeStop_active : BOOL := FALSE;
  Branch_0_active : BOOL := FALSE;
  Branch_1_active : BOOL := FALSE;
  Branch_2_active : BOOL := FALSE;
  Step_255_active : BOOL := FALSE;
  ApplyOutput_active : BOOL := FALSE;
  SafetyInputMonitor_active : BOOL := FALSE;
  SafetyLog_active : BOOL := FALSE;
  IN : INT := 0;
  TEST : INT := 0;
  ARE : INT := 0;
  CYCLE_TIME : TIME := T#0s;
  SENS : INT := 0;
  SELF_ACT_TIME : TIME := T#0s;
  SELF_ACT_PULSE : TIME := T#0s;
  SELF_ACT_CYCLES : INT := 0;
  OUT : BOOL := FALSE;
  ARO : BOOL := FALSE;
  ARX : INT := 0;
  timer : TIMER;
  pwgen : PWGEN;
  InputValidFlag : BOOL := FALSE;
  SafetyErrorFlag : BOOL := FALSE;
  SafetyErrorActive : BOOL := FALSE;
  TimeoutErrorFlag : BOOL := FALSE;
  SafetyCycleCounter : INT := 0;
  SafetyResetCommand : BOOL := FALSE;
  TimeoutResetCommand : BOOL := FALSE;
  MonitorValidFlag : BOOL := FALSE;
  LastCycleCounter : INT := 0;
  LastErrorState : BOOL := FALSE;
END_VAR

(* --- Initialize initial step --- *)
IF NOT InitCycle_active THEN
  InitCycle_active := TRUE;
END_IF;

(* --- Step actions --- *)
IF InitCycle_active THEN
  timer(trun := MUL_T_AI(SELF_ACT_PULSE,2 * SELF_ACT_CYCLES), toff := SELF_ACT_TIME, Test := TEST, ARE := ARE, arx := ARX); ARX := timer.ARX; ARO := timer.ARO; SafetyCycleCounter := SafetyCycleCounter + 1;
END_IF;
IF SafetyCheckInput_active THEN
  InputValidFlag := (IN >= BYTE#0) AND (IN <= BYTE#255) AND (SENS > BYTE#0) AND (SENS <= BYTE#255); SafetyErrorFlag := NOT InputValidFlag;
END_IF;
IF SafetyError_active THEN
  out := FALSE; SafetyErrorActive := TRUE; ARO := FALSE;
END_IF;
IF TimeoutSafeStop_active THEN
  out := FALSE; TimeoutErrorFlag := TRUE; ARO := FALSE; SafetyCycleCounter := 0;
END_IF;
IF Branch_0_active THEN
  pwgen(PTL := SELF_ACT_PULSE, PTH := SELF_ACT_PULSE); out := pwgen.Q;
END_IF;
IF Branch_1_active THEN
  out := FALSE;
END_IF;
IF Branch_2_active THEN
  out := TRUE;
END_IF;
IF Step_255_active THEN
  pwgen.PTH := (CYCLE_TIME * BYTE_TO_TIME(BAND_B(IN,SENS)) ) / BYTE_TO_TIME(BYTE#255); pwgen.PTL := CYCLE_TIME - pwgen.PTH; pwgen(); out := pwgen.Q;
END_IF;
IF SafetyInputMonitor_active THEN
  MonitorValidFlag := (IN >= BYTE#0) AND (IN <= BYTE#255) AND (SENS > BYTE#0) AND (SENS <= BYTE#255);
END_IF;
IF SafetyLog_active THEN
  LastCycleCounter := SafetyCycleCounter; LastErrorState := SafetyErrorActive OR TimeoutErrorFlag;
END_IF;

(* --- Transitions --- *)
IF InitCycle_active AND (TRUE) THEN
  InitCycle_active := FALSE;
  SafetyCheckInput_active := TRUE;
END_IF;
IF InitCycle_active AND (TRUE) THEN
  InitCycle_active := FALSE;
  SafetyInputMonitor_active := TRUE;
END_IF;
IF SafetyInputMonitor_active AND (MonitorValidFlag = FALSE) THEN
  SafetyInputMonitor_active := FALSE;
  SafetyError_active := TRUE;
END_IF;
IF SafetyInputMonitor_active AND (MonitorValidFlag = TRUE) THEN
  SafetyInputMonitor_active := FALSE;
  SafetyInputMonitor_active := TRUE;
END_IF;
IF SafetyCheckInput_active AND (SafetyErrorFlag = TRUE) THEN
  SafetyCheckInput_active := FALSE;
  SafetyError_active := TRUE;
END_IF;
IF SafetyCheckInput_active AND (SafetyErrorFlag = FALSE AND SafetyCycleCounter > (SELF_ACT_CYCLES * 3)) THEN
  SafetyCheckInput_active := FALSE;
  TimeoutSafeStop_active := TRUE;
END_IF;
IF SafetyCheckInput_active AND (SafetyErrorFlag = FALSE AND SafetyCycleCounter <= (SELF_ACT_CYCLES * 3) AND aro = TRUE) THEN
  SafetyCheckInput_active := FALSE;
  Branch_0_active := TRUE;
END_IF;
IF SafetyCheckInput_active AND (SafetyErrorFlag = FALSE AND SafetyCycleCounter <= (SELF_ACT_CYCLES * 3) AND aro = FALSE AND in<sens) THEN
  SafetyCheckInput_active := FALSE;
  Branch_1_active := TRUE;
END_IF;
IF SafetyCheckInput_active AND (SafetyErrorFlag = FALSE AND SafetyCycleCounter <= (SELF_ACT_CYCLES * 3) AND aro = FALSE AND NOT (in<sens) AND BYTE_TO_USINT(in)>USINT#255-BYTE_TO_USINT(sens)) THEN
  SafetyCheckInput_active := FALSE;
  Branch_2_active := TRUE;
END_IF;
IF SafetyCheckInput_active AND (SafetyErrorFlag = FALSE AND SafetyCycleCounter <= (SELF_ACT_CYCLES * 3) AND aro = FALSE AND NOT (in<sens) AND NOT (BYTE_TO_USINT(in)>USINT#255-BYTE_TO_USINT(sens))) THEN
  SafetyCheckInput_active := FALSE;
  Step_255_active := TRUE;
END_IF;
IF Branch_0_active AND (TRUE) THEN
  Branch_0_active := FALSE;
  ApplyOutput_active := TRUE;
END_IF;
IF Branch_1_active AND (TRUE) THEN
  Branch_1_active := FALSE;
  ApplyOutput_active := TRUE;
END_IF;
IF Branch_2_active AND (TRUE) THEN
  Branch_2_active := FALSE;
  ApplyOutput_active := TRUE;
END_IF;
IF Step_255_active AND (TRUE) THEN
  Step_255_active := FALSE;
  ApplyOutput_active := TRUE;
END_IF;
IF ApplyOutput_active AND (SafetyErrorActive = FALSE AND TimeoutErrorFlag = FALSE) THEN
  ApplyOutput_active := FALSE;
  SafetyLog_active := TRUE;
END_IF;
IF SafetyLog_active AND (TRUE) THEN
  SafetyLog_active := FALSE;
  InitCycle_active := TRUE;
END_IF;
IF SafetyError_active AND (SafetyResetCommand = TRUE) THEN
  SafetyError_active := FALSE;
  InitCycle_active := TRUE;
END_IF;
IF TimeoutSafeStop_active AND (TimeoutResetCommand = TRUE) THEN
  TimeoutSafeStop_active := FALSE;
  InitCycle_active := TRUE;
END_IF;

END_PROGRAM

(* ---- ACTUATOR_2P_sfc_iter_03_upgraded.st ---- *)
PROGRAM SFC_Program
(* Auto-generated by SFCJSONConverter *)

VAR
  InitCycle_active : BOOL := FALSE;
  SafetyCheckInput_active : BOOL := FALSE;
  SafetyError_active : BOOL := FALSE;
  TimeoutSafeStop_active : BOOL := FALSE;
  Branch_0_active : BOOL := FALSE;
  Branch_1_active : BOOL := FALSE;
  Branch_2_active : BOOL := FALSE;
  Step_255_active : BOOL := FALSE;
  ApplyOutput_active : BOOL := FALSE;
  IN : INT := 0;
  TEST : INT := 0;
  ARE : INT := 0;
  CYCLE_TIME : TIME := T#0s;
  SENS : INT := 0;
  SELF_ACT_TIME : TIME := T#0s;
  SELF_ACT_PULSE : TIME := T#0s;
  SELF_ACT_CYCLES : INT := 0;
  OUT : BOOL := FALSE;
  ARO : BOOL := FALSE;
  ARX : INT := 0;
  timer : TIMER;
  pwgen : PWGEN;
  InputValidFlag : BOOL := FALSE;
  SafetyErrorFlag : BOOL := FALSE;
  SafetyErrorActive : BOOL := FALSE;
  TimeoutErrorFlag : BOOL := FALSE;
  SafetyCycleCounter : INT := 0;
  SafetyResetCommand : BOOL := FALSE;
  TimeoutResetCommand : BOOL := FALSE;
END_VAR

(* --- Initialize initial step --- *)
IF NOT InitCycle_active THEN
  InitCycle_active := TRUE;
END_IF;

(* --- Step actions --- *)
IF InitCycle_active THEN
  timer(trun := MUL_T_AI(SELF_ACT_PULSE,2 * SELF_ACT_CYCLES), toff := SELF_ACT_TIME, Test := TEST, ARE := ARE, arx := ARX); ARX := timer.ARX; ARO := timer.ARO; SafetyCycleCounter := SafetyCycleCounter + 1;
END_IF;
IF SafetyCheckInput_active THEN
  InputValidFlag := (IN >= BYTE#0) AND (IN <= BYTE#255) AND (SENS > BYTE#0) AND (SENS <= BYTE#255); SafetyErrorFlag := NOT InputValidFlag;
END_IF;
IF SafetyError_active THEN
  out := FALSE; SafetyErrorActive := TRUE; ARO := FALSE;
END_IF;
IF TimeoutSafeStop_active THEN
  out := FALSE; TimeoutErrorFlag := TRUE; ARO := FALSE; SafetyCycleCounter := 0;
END_IF;
IF Branch_0_active THEN
  pwgen(PTL := SELF_ACT_PULSE, PTH := SELF_ACT_PULSE); out := pwgen.Q;
END_IF;
IF Branch_1_active THEN
  out := FALSE;
END_IF;
IF Branch_2_active THEN
  out := TRUE;
END_IF;
IF Step_255_active THEN
  pwgen.PTH := (CYCLE_TIME * BYTE_TO_TIME(BAND_B(IN,SENS)) ) / BYTE_TO_TIME(BYTE#255); pwgen.PTL := CYCLE_TIME - pwgen.PTH; pwgen(); out := pwgen.Q;
END_IF;

(* --- Transitions --- *)
IF InitCycle_active AND (TRUE) THEN
  InitCycle_active := FALSE;
  SafetyCheckInput_active := TRUE;
END_IF;
IF SafetyCheckInput_active AND (SafetyErrorFlag = TRUE) THEN
  SafetyCheckInput_active := FALSE;
  SafetyError_active := TRUE;
END_IF;
IF SafetyCheckInput_active AND (SafetyErrorFlag = FALSE AND SafetyCycleCounter > (SELF_ACT_CYCLES * 3)) THEN
  SafetyCheckInput_active := FALSE;
  TimeoutSafeStop_active := TRUE;
END_IF;
IF SafetyCheckInput_active AND (SafetyErrorFlag = FALSE AND SafetyCycleCounter <= (SELF_ACT_CYCLES * 3) AND aro = TRUE) THEN
  SafetyCheckInput_active := FALSE;
  Branch_0_active := TRUE;
END_IF;
IF SafetyCheckInput_active AND (SafetyErrorFlag = FALSE AND SafetyCycleCounter <= (SELF_ACT_CYCLES * 3) AND aro = FALSE AND in<sens) THEN
  SafetyCheckInput_active := FALSE;
  Branch_1_active := TRUE;
END_IF;
IF SafetyCheckInput_active AND (SafetyErrorFlag = FALSE AND SafetyCycleCounter <= (SELF_ACT_CYCLES * 3) AND aro = FALSE AND NOT (in<sens) AND BYTE_TO_USINT(in)>USINT#255-BYTE_TO_USINT(sens)) THEN
  SafetyCheckInput_active := FALSE;
  Branch_2_active := TRUE;
END_IF;
IF SafetyCheckInput_active AND (SafetyErrorFlag = FALSE AND SafetyCycleCounter <= (SELF_ACT_CYCLES * 3) AND aro = FALSE AND NOT (in<sens) AND NOT (BYTE_TO_USINT(in)>USINT#255-BYTE_TO_USINT(sens))) THEN
  SafetyCheckInput_active := FALSE;
  Step_255_active := TRUE;
END_IF;
IF Branch_0_active AND (TRUE) THEN
  Branch_0_active := FALSE;
  ApplyOutput_active := TRUE;
END_IF;
IF Branch_1_active AND (TRUE) THEN
  Branch_1_active := FALSE;
  ApplyOutput_active := TRUE;
END_IF;
IF Branch_2_active AND (TRUE) THEN
  Branch_2_active := FALSE;
  ApplyOutput_active := TRUE;
END_IF;
IF Step_255_active AND (TRUE) THEN
  Step_255_active := FALSE;
  ApplyOutput_active := TRUE;
END_IF;
IF ApplyOutput_active AND (SafetyErrorActive = FALSE AND TimeoutErrorFlag = FALSE) THEN
  ApplyOutput_active := FALSE;
  InitCycle_active := TRUE;
END_IF;
IF SafetyError_active AND (SafetyResetCommand = TRUE) THEN
  SafetyError_active := FALSE;
  InitCycle_active := TRUE;
END_IF;
IF TimeoutSafeStop_active AND (TimeoutResetCommand = TRUE) THEN
  TimeoutSafeStop_active := FALSE;
  InitCycle_active := TRUE;
END_IF;

END_PROGRAM
